// TIA Portal project "HIDROCONTROL" (V17)

(* hardware
DEVICE "S7-1200 station_1"  S7-1200 Station
   slot 0: "Rack_0"  S7-1200 Rack  Rack  V1.0
   slot 1: "PLC_1"  CPU 1214C AC/DC/Rly  6ES7 214-1BG40-0XB0  V4.5
*)

// ===== PLC "PLC_1"  CPU 1214C AC/DC/Rly =====

VAR_GLOBAL   // PLC tag table "Default tag table"
   "Clock_Byte" AT %MB0 : Byte;
   "Clock_10Hz" AT %M0.0 : Bool;
   "Clock_5Hz" AT %M0.1 : Bool;
   "Clock_2.5Hz" AT %M0.2 : Bool;
   "Clock_2Hz" AT %M0.3 : Bool;
   "Clock_1.25Hz" AT %M0.4 : Bool;
   "Clock_1Hz" AT %M0.5 : Bool;
   "Clock_0.625Hz" AT %M0.6 : Bool;
   "Clock_0.5Hz" AT %M0.7 : Bool;
   "Tag_1" AT %M10.0 : Bool;
   "Tag_2" AT %Q0.0 : Bool;
   "B1" AT %Q0.1 : Bool;
   "Tag_3" AT %Q0.2 : Bool;
   "Tag_4" AT %Q0.3 : Bool;
   "Tag_5" AT %I0.0 : Bool;
   "Tag_6" AT %IW64 : Int;
   "Tag_7" AT %MD2 : Real;
   "tag_8" AT %MD6 : Real;
   "tag_9" AT %MD12 : Real;
   "tag_10" AT %MD16 : Real;
END_VAR

DATA_BLOCK "DB10_SCADA_READ"   // DB10
{ S7_Optimized_Access := 'FALSE' }
VERSION : 0.1
   VAR
      bomba_principal_estado : Bool;   // Estado real B1
      dosificador_sulfato_estado : Bool;   // Estado real B2
      dosificador_cloro_estado : Bool;   // Estado real B3
      nivel_tanque_agua_cruda : Bool;   // Sensor digital nivel S1
      modo_remoto_habilitado : Bool;   // Permite comandos remotos
      plc_en_falla : Bool;   // Falla general PLC/proceso
      comando_rechazado : Bool;   // PLC rechazo ultimo comando
      ultimo_comando_aceptado : Bool;   // PLC acepto ultimo comando
      ph_agua_cruda : Real;   // S2 escalado en pH
      turbidez_agua_cruda : Real;   // S3 escalado en NTU
      conductividad_agua_cruda : Real;   // S4 escalado en uS/cm
      ph_agua_tratada : Real;   // S5 escalado en pH
      turbidez_agua_tratada : Real;   // S6 escalado en NTU
      conductividad_agua_tratada : Real;   // S7 escalado en uS/cm
      caudal_bomba_principal : Real;   // S8 escalado en L/min
      caudal_distribucion : Real;   // S9 escalado en L/min
      presion_bomba_principal : Real;   // S10 escalado en bar, pendiente canal fisico
      watchdog_plc : DInt;   // Contador vivo desde PLC
   END_VAR
BEGIN
END_DATA_BLOCK

DATA_BLOCK "DB11_SCADA_WRITE"   // DB11
{ S7_Optimized_Access := 'FALSE' }
VERSION : 0.1
   VAR
      comando_bomba_principal_start : Bool;   // comando_bomba_principal_start
      comando_bomba_principal_stop : Bool;   // comando_bomba_principal_stop
      comando_dosificador_sulfato_start : Bool;   // comando_dosificador_sulfato_start
      comando_dosificador_sulfato_stop : Bool;   // comando_dosificador_sulfato_stop
      comando_dosificador_cloro_start : Bool;   // comando_dosificador_cloro_start
      comando_dosificador_cloro_stop : Bool;   // comando_dosificador_cloro_stop
      reset_alarmas : Bool;   // reset_alarmas
      watchdog_scada : Bool;   // watchdog_scada
      command_sequence : DInt;   // command_sequence
   END_VAR
BEGIN
END_DATA_BLOCK

ORGANIZATION_BLOCK "Main"   // OB1, LAD, ProgramCycle
TITLE = "Main Program Sweep (Cycle)"
{ S7_Optimized_Access := 'TRUE' }
VERSION : 0.1
   VAR_INPUT
      Initial_Call : Bool;   // Initial call of this OB
      Remanence : Bool;   // =True, if remanent data are available
   END_VAR
   VAR_TEMP   // added for the SCL form of the ladder/FBD networks
      _w1 : Bool;
   END_VAR
BEGIN

REGION Network 1: Prender B1
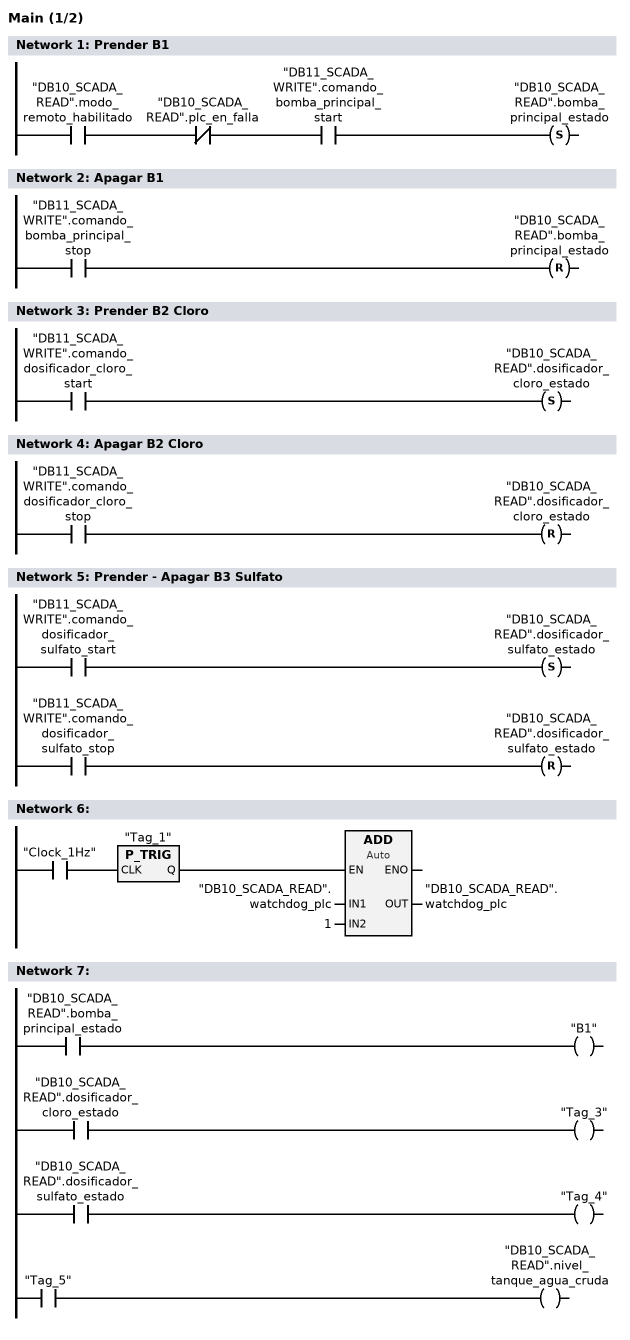
   RUNG wire#powerrail
      Contact( "DB10_SCADA_READ".modo_remoto_habilitado )
      I_Contact( "DB10_SCADA_READ".plc_en_falla )
      Contact( "DB11_SCADA_WRITE".comando_bomba_principal_start )
      S_Coil( "DB10_SCADA_READ".bomba_principal_estado )
   END_RUNG
   // the same network as SCL:
   IF "DB10_SCADA_READ".modo_remoto_habilitado AND NOT "DB10_SCADA_READ".plc_en_falla AND "DB11_SCADA_WRITE".comando_bomba_principal_start THEN
       "DB10_SCADA_READ".bomba_principal_estado := TRUE;
   END_IF;
END_REGION

REGION Network 2: Apagar B1
   RUNG wire#powerrail
      Contact( "DB11_SCADA_WRITE".comando_bomba_principal_stop )
      R_Coil( "DB10_SCADA_READ".bomba_principal_estado )
   END_RUNG
   // the same network as SCL:
   IF "DB11_SCADA_WRITE".comando_bomba_principal_stop THEN
       "DB10_SCADA_READ".bomba_principal_estado := FALSE;
   END_IF;
END_REGION

REGION Network 3: Prender B2 Cloro
   RUNG wire#powerrail
      Contact( "DB11_SCADA_WRITE".comando_dosificador_cloro_start )
      S_Coil( "DB10_SCADA_READ".dosificador_cloro_estado )
   END_RUNG
   // the same network as SCL:
   IF "DB11_SCADA_WRITE".comando_dosificador_cloro_start THEN
       "DB10_SCADA_READ".dosificador_cloro_estado := TRUE;
   END_IF;
END_REGION

REGION Network 4: Apagar B2 Cloro
   RUNG wire#powerrail
      Contact( "DB11_SCADA_WRITE".comando_dosificador_cloro_stop )
      R_Coil( "DB10_SCADA_READ".dosificador_cloro_estado )
   END_RUNG
   // the same network as SCL:
   IF "DB11_SCADA_WRITE".comando_dosificador_cloro_stop THEN
       "DB10_SCADA_READ".dosificador_cloro_estado := FALSE;
   END_IF;
END_REGION

REGION Network 5: Prender - Apagar B3 Sulfato
   RUNG wire#powerrail
      Contact( "DB11_SCADA_WRITE".comando_dosificador_sulfato_start )
      S_Coil( "DB10_SCADA_READ".dosificador_sulfato_estado )
   END_RUNG
   RUNG wire#powerrail
      Contact( "DB11_SCADA_WRITE".comando_dosificador_sulfato_stop )
      R_Coil( "DB10_SCADA_READ".dosificador_sulfato_estado )
   END_RUNG
   // the same network as SCL:
   IF "DB11_SCADA_WRITE".comando_dosificador_sulfato_start THEN
       "DB10_SCADA_READ".dosificador_sulfato_estado := TRUE;
   END_IF;
   IF "DB11_SCADA_WRITE".comando_dosificador_sulfato_stop THEN
       "DB10_SCADA_READ".dosificador_sulfato_estado := FALSE;
   END_IF;
END_REGION

REGION Network 6
   RUNG wire#powerrail
      Contact( "Clock_1Hz" )
      P_Trig( "Tag_1" )
      Add(in1 := "DB10_SCADA_READ".watchdog_plc, in2 := 1, out => "DB10_SCADA_READ".watchdog_plc)
   END_RUNG
   // the same network as SCL:
   #_w1 := "Clock_1Hz" AND NOT "Tag_1";   // rising edge
   "Tag_1" := "Clock_1Hz";
   IF #_w1 THEN "DB10_SCADA_READ".watchdog_plc := "DB10_SCADA_READ".watchdog_plc + 1; END_IF;
END_REGION

REGION Network 7
   RUNG wire#powerrail
      Contact( "DB10_SCADA_READ".bomba_principal_estado )
      Coil( "B1" )
   END_RUNG
   RUNG wire#powerrail
      Contact( "DB10_SCADA_READ".dosificador_cloro_estado )
      Coil( "Tag_3" )
   END_RUNG
   RUNG wire#powerrail
      Contact( "DB10_SCADA_READ".dosificador_sulfato_estado )
      Coil( "Tag_4" )
   END_RUNG
   RUNG wire#powerrail
      Contact( "Tag_5" )
      Coil( "DB10_SCADA_READ".nivel_tanque_agua_cruda )
   END_RUNG
   // the same network as SCL:
   "B1" := "DB10_SCADA_READ".bomba_principal_estado;
   "Tag_3" := "DB10_SCADA_READ".dosificador_cloro_estado;
   "Tag_4" := "DB10_SCADA_READ".dosificador_sulfato_estado;
   "DB10_SCADA_READ".nivel_tanque_agua_cruda := "Tag_5";
END_REGION

REGION Network 8
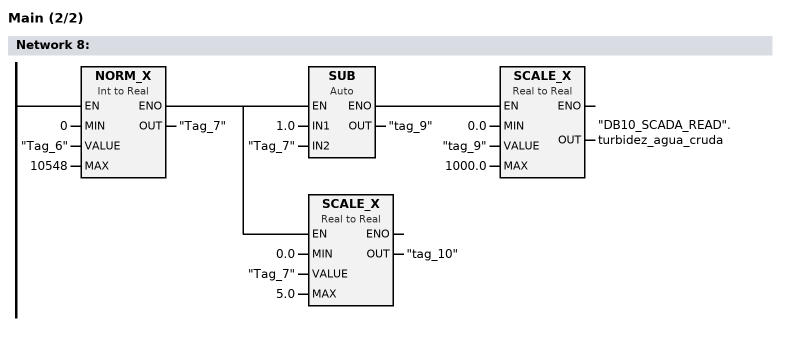
   RUNG wire#powerrail
      { S7_Templates := "[SrcType := Int, DestType := Real]" } Normalize(min := 0, value := "Tag_6", max := 10548, out => "Tag_7")
      wire#w1
      Sub(in1 := 1.0, in2 := "Tag_7", out => "tag_9")
      { S7_Templates := "[SrcType := Real, DestType := Real]" } Scale(min := 0.0, value := "tag_9", max := 1000.0, out => "DB10_SCADA_READ".turbidez_agua_cruda)
   END_RUNG
   RUNG wire#w1
      { S7_Templates := "[SrcType := Real, DestType := Real]" } Scale(min := 0.0, value := "Tag_7", max := 5.0, out => "tag_10")
   END_RUNG
   // the same network as SCL:
   "Tag_7" := NORM_X(MIN := 0, VALUE := "Tag_6", MAX := 10548);
   "tag_9" := 1.0 - "Tag_7";
   "DB10_SCADA_READ".turbidez_agua_cruda := SCALE_X(MIN := 0.0, VALUE := "tag_9", MAX := 1000.0);
   "tag_10" := SCALE_X(MIN := 0.0, VALUE := "Tag_7", MAX := 5.0);
END_REGION
END_ORGANIZATION_BLOCK